# EPICS substitutions: db/Beckhoff_3XXX/ecmcEP3162.substitutions
# analog inputs
file "ecmc_analogInput-chX.template"{
  pattern {CH_ID, ESLO, EOFF, EGU, PREC}
          {01, "${_ESLO=3.0518509476E-4}", "${_EOFF=0}", "${_EGU=V}", "${_PREC=3}"}
          {02, "${_ESLO=3.0518509476E-4}", "${_EOFF=0}", "${_EGU=V}", "${_PREC=3}"}
}

# channel status
file "ecmc_status_analog-chX.template"{
  pattern {CH_ID, KEY}
          {01,    AI }
          {02,    AI }
}
